Yaskawa INFORM job: BATMAN_ALL.JBI

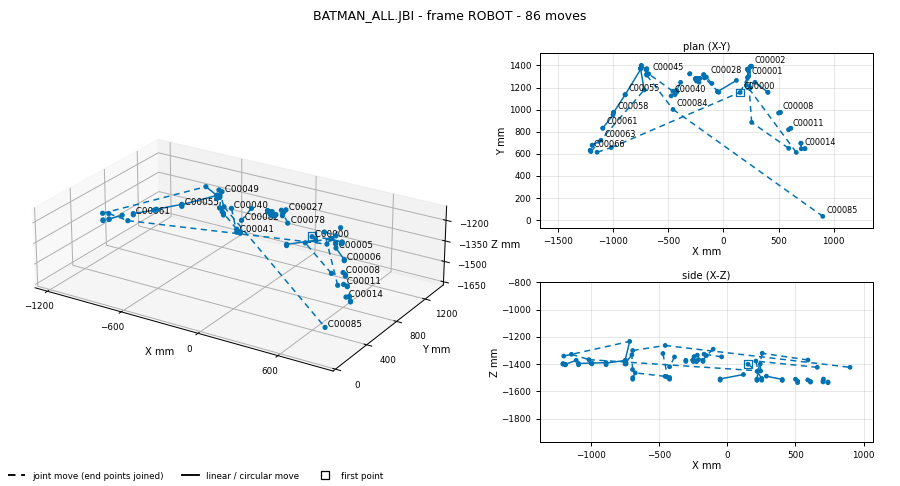
[picture p0: tool path of BATMAN_ALL.JBI in frame ROBOT, 86 of 157 moves have a stored position in this frame; points joined in program order, loops and branches not executed]
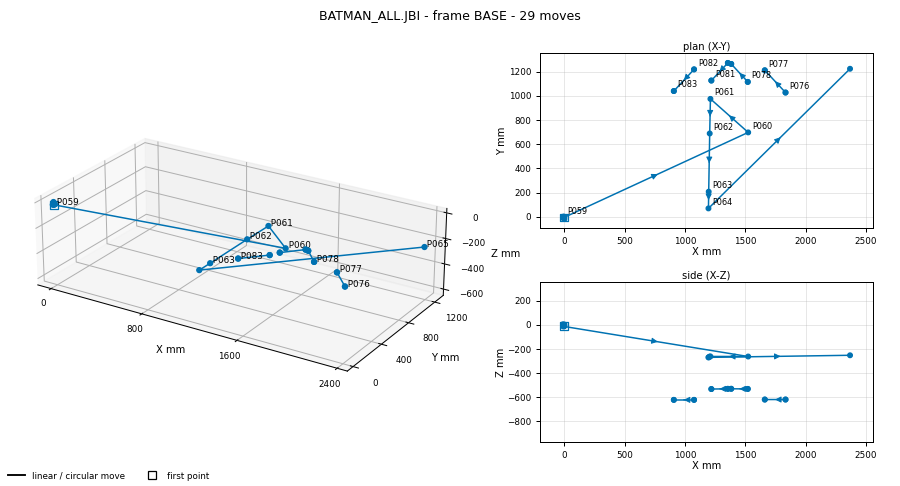
[picture p1: tool path of BATMAN_ALL.JBI in frame BASE, 29 of 157 moves have a stored position in this frame; points joined in program order, loops and branches not executed]
/JOB
//NAME BATMAN_ALL
///FOLDERNAME KRIS-SCIANA
//POS
///NPOS 86,86,0,38,0,0
///TOOL 0
///POSTYPE ROBOT
///RECTAN
///RCONF 0,0,0,0,0,0,0,0,0,0,0,0,0,0,0,0,0,0,0,0,0,0,0,0
C00000=152.410,1154.783,-1401.344,10.8585,26.8248,-46.4937
C00001=219.135,1290.433,-1453.397,13.1324,27.7106,-79.4132
C00002=252.850,1392.626,-1506.056,13.1307,27.7072,-79.4089
C00003=252.842,1392.620,-1508.783,13.1301,27.7068,-79.4080
C00004=252.850,1392.613,-1518.378,13.1306,27.7064,-79.4089
C00005=287.081,1247.667,-1488.936,13.1308,27.7079,-79.4066
C00006=403.589,1157.140,-1512.613,13.1304,27.7106,-79.4046
C00007=403.589,1157.122,-1519.985,13.1305,27.7097,-79.4043
C00008=500.680,969.258,-1511.018,13.1325,27.7074,-79.4005
C00009=516.044,974.881,-1524.930,13.1331,27.7092,-79.4004
C00010=516.045,974.868,-1535.811,13.1328,27.7077,-79.4001
C00011=590.606,818.366,-1515.976,13.1319,27.7058,-79.3988
C00012=610.782,831.337,-1527.481,13.1332,27.7070,-79.3997
C00013=610.774,831.333,-1532.290,13.1329,27.7070,-79.3992
C00014=705.770,645.699,-1509.934,13.1296,27.7061,-79.4018
C00015=702.820,695.837,-1524.665,13.1293,27.7044,-79.3984
C00016=702.809,695.833,-1530.916,13.1291,27.7040,-79.3963
C00017=738.969,646.930,-1531.718,13.1275,27.7068,-79.4007
C00018=738.965,646.937,-1536.801,13.1273,27.7075,-79.4010
C00019=592.006,649.855,-1370.263,13.1298,27.7033,-79.3961
C00020=256.954,884.347,-1320.582,10.9643,26.7399,-79.4986
C00021=226.416,1297.769,-1450.356,10.9643,26.7388,-15.7591
C00022=218.104,1365.766,-1510.694,4.6590,27.3838,-18.5852
C00023=218.092,1365.754,-1519.334,4.6575,27.3846,-18.5871
C00024=118.975,1264.663,-1476.628,4.6556,27.3863,-18.5969
C00025=-51.918,1162.894,-1508.930,4.6554,27.3843,-18.5935
C00026=-51.924,1162.893,-1518.207,4.6552,27.3847,-18.5926
C00027=-103.106,1236.815,-1291.023,4.6548,27.3832,-18.5938
C00028=-153.186,1294.382,-1337.444,-2.5810,29.3407,-40.5711
C00029=-177.451,1316.167,-1372.170,-2.5797,29.3412,-40.5749
C00030=-177.463,1316.142,-1380.653,-2.5821,29.3407,-40.5765
C00031=-210.259,1283.024,-1367.501,-2.5843,29.3397,-40.5838
C00032=-225.620,1283.017,-1376.307,-2.5829,29.3396,-40.5802
C00033=-225.613,1283.030,-1382.225,-2.5820,29.3397,-40.5809
C00034=-243.196,1259.338,-1345.105,-2.5829,29.3386,-40.5814
C00035=-253.627,1276.795,-1370.708,-2.5815,29.3400,-94.0341
C00036=-248.341,1281.400,-1375.363,-2.5806,29.3383,-94.0334
C00037=-248.343,1281.405,-1380.636,-2.5812,29.3384,-94.0354
C00038=-303.361,1324.266,-1372.348,-2.5804,29.3359,-94.0344
C00039=-303.363,1324.269,-1380.668,-2.5806,29.3358,-94.0352
C00040=-471.541,1124.138,-1322.421,-2.5821,29.3374,-94.0378
C00041=-436.993,1135.677,-1497.127,-2.5833,29.3385,-94.0377
C00042=-422.594,1159.988,-1498.740,-2.5814,29.3381,-94.0327
C00043=-422.595,1159.986,-1510.903,-2.5817,29.3385,-94.0330
C00044=-455.700,1166.055,-1490.114,-2.5799,29.3369,-94.0339
C00045=-674.596,1323.179,-1464.338,-2.5825,29.3370,-94.0343
C00046=-692.829,1369.142,-1499.740,-2.5956,29.3274,-94.0386
C00047=-692.829,1369.134,-1511.111,-2.5953,29.3273,-94.0360
C00048=-694.274,1320.333,-1440.373,-2.5948,29.3272,-94.0370
C00049=-699.144,1360.561,-1331.781,19.2113,25.3199,54.7614
C00050=-742.001,1399.272,-1388.079,19.2141,25.3197,54.7634
C00051=-742.001,1399.307,-1398.942,19.2156,25.3171,54.7657
C00052=-749.229,1371.947,-1375.142,19.2122,25.3194,54.7649
C00053=-749.245,1371.950,-1399.047,19.2137,25.3200,54.7650
C00054=-744.062,1371.872,-1373.000,19.2081,25.3216,54.7703
C00055=-888.177,1135.095,-1392.458,19.2114,25.3213,54.7713
C00056=-888.162,1135.097,-1404.947,19.2099,25.3206,54.7706
C00057=-888.146,1135.084,-1389.652,19.2087,25.3204,54.7704
C00058=-992.935,974.707,-1392.448,19.2118,25.3202,54.7709
C00059=-992.926,974.691,-1398.054,19.2108,25.3207,54.7707
C00060=-998.229,951.939,-1392.438,19.2128,25.3209,54.7710
C00061=-1090.439,832.216,-1395.757,19.2120,25.3253,54.7669
C00062=-1090.449,832.216,-1404.874,19.2124,25.3260,54.7666
C00063=-1107.538,722.615,-1372.300,19.2115,25.3258,54.7652
C00064=-1186.713,677.650,-1401.899,19.2118,25.3233,54.7691
C00065=-1186.711,677.656,-1405.576,19.2118,25.3228,54.7692
C00066=-1204.504,631.027,-1396.106,19.2134,25.3226,54.7707
C00067=-1204.501,631.029,-1401.004,19.2135,25.3224,54.7708
C00068=-1198.537,620.359,-1341.276,19.2108,25.3216,54.7720
C00069=-715.412,1179.070,-1233.819,19.2159,25.3335,54.7762
C00070=-749.229,1371.947,-1375.142,19.2122,25.3194,54.7649
C00071=-1142.143,614.362,-1328.458,18.1291,25.2802,54.3071
C00072=-1014.182,656.385,-1367.467,19.2126,25.3035,24.7793
C00073=244.678,1197.356,-1450.442,14.1934,24.5334,-60.4282
C00074=242.567,1385.701,-1399.440,12.9652,27.2001,-79.4839
C00075=660.569,613.161,-1423.808,13.1448,27.7005,-139.3923
C00076=210.374,1220.455,-1377.909,14.2177,19.9635,-61.8713
C00077=226.382,1351.810,-1450.861,14.2179,19.9642,-61.8758
C00078=-41.244,1157.338,-1346.763,4.6551,27.3861,-18.5879
C00079=-169.787,1287.439,-1327.342,-2.5927,29.3373,-40.6168
C00080=-219.530,1247.683,-1334.789,-2.5902,29.3364,-82.5753
C00081=-386.471,1247.154,-1347.732,14.2186,19.9661,-61.8751
C00082=-422.753,1176.097,-1419.836,-2.5966,29.3308,-94.0443
C00083=-692.993,1311.701,-1300.606,-2.6070,29.3169,-94.0355
C00084=-454.695,1001.750,-1263.493,10.2829,30.0776,-90.6322
C00085=900.646,33.952,-1423.808,13.1448,27.7005,179.8982
BC00000=1473.101,32.856,1458.546
BC00001=1602.629,32.856,1262.258
BC00002=1602.629,32.863,1262.252
BC00003=1602.629,32.863,1262.252
BC00004=1602.629,32.863,1262.252
BC00005=1602.629,32.863,1262.252
BC00006=1602.629,32.863,1262.248
BC00007=1602.629,32.863,1262.248
BC00008=1602.629,32.863,1262.248
BC00009=1602.629,32.863,1262.248
BC00010=1602.629,32.863,1262.248
BC00011=1602.629,32.863,1262.248
BC00012=1602.629,32.863,1262.248
BC00013=1602.629,32.863,1262.248
BC00014=1602.629,32.863,1262.248
BC00015=1602.629,32.863,1262.248
BC00016=1602.629,32.863,1262.248
BC00017=1602.629,32.863,1262.248
BC00018=1602.629,32.863,1262.248
BC00019=1602.629,32.863,1262.248
BC00020=1602.629,32.863,1262.248
BC00021=1602.629,32.863,1262.248
BC00022=1602.629,32.863,1262.248
BC00023=1602.629,32.863,1262.248
BC00024=1602.629,32.863,1262.248
BC00025=1602.629,32.863,1262.248
BC00026=1602.629,32.863,1262.248
BC00027=1602.629,32.863,1262.248
BC00028=1602.629,32.863,1262.248
BC00029=1602.629,32.863,1262.248
BC00030=1602.629,32.863,1262.248
BC00031=1602.629,32.863,1262.248
BC00032=1602.629,32.863,1262.248
BC00033=1602.629,32.863,1262.248
BC00034=1602.629,32.863,1262.248
BC00035=1602.629,32.863,1262.248
BC00036=1602.629,32.863,1262.248
BC00037=1602.629,32.863,1262.248
BC00038=1602.629,32.863,1262.248
BC00039=1602.629,32.863,1262.248
BC00040=1602.629,32.863,1262.248
BC00041=1602.629,32.863,1262.248
BC00042=1602.629,32.863,1262.248
BC00043=1602.629,32.863,1262.248
BC00044=1602.629,32.863,1262.248
BC00045=1602.629,32.863,1262.248
BC00046=1602.623,32.869,1262.243
BC00047=1602.623,32.869,1262.243
BC00048=1602.623,32.869,1262.243
BC00049=1602.629,32.850,1148.408
BC00050=1602.629,32.850,1148.408
BC00051=1602.629,32.850,1148.408
BC00052=1602.629,32.850,1148.408
BC00053=1602.629,32.850,1148.408
BC00054=1602.629,32.850,1148.408
BC00055=1602.629,32.850,1148.408
BC00056=1602.629,32.850,1148.408
BC00057=1602.629,32.850,1148.408
BC00058=1602.629,32.850,1148.408
BC00059=1602.629,32.850,1148.408
BC00060=1602.629,32.850,1148.408
BC00061=1602.629,32.850,1148.408
BC00062=1602.629,32.850,1148.408
BC00063=1602.629,32.850,1148.408
BC00064=1602.629,32.850,1148.408
BC00065=1602.629,32.850,1148.408
BC00066=1602.629,32.850,1148.408
BC00067=1602.629,32.850,1148.408
BC00068=1602.629,32.850,1148.408
BC00069=1602.629,32.856,1148.402
BC00070=1602.629,32.850,1148.408
BC00071=1602.629,32.850,1148.408
BC00072=1602.629,32.856,1527.186
BC00073=1602.629,32.856,1413.595
BC00074=1602.629,32.863,1262.252
BC00075=1602.629,32.863,1262.252
BC00076=1602.629,32.863,1262.252
BC00077=1602.629,32.863,1262.252
BC00078=1602.629,32.863,1262.252
BC00079=1602.629,32.863,1262.252
BC00080=1602.629,32.863,1262.252
BC00081=1602.629,32.863,1262.252
BC00082=1602.629,32.863,1262.252
BC00083=1602.629,32.863,1262.252
BC00084=1602.629,32.863,1262.252
BC00085=899.093,32.863,1856.752
///POSTYPE BASE
P00059=-2.448,-6.714,-12.718,0.0000,0.0000,0.0000
P00060=1524.284,698.404,-261.973,-0.4635,36.8346,-1.2388
P00061=1211.499,975.999,-261.374,0.5148,35.2356,175.5099
P00062=1205.574,689.500,-262.704,0.5159,35.2461,175.5270
P00063=1197.217,207.358,-268.729,0.4863,35.2395,175.4586
P00064=1195.199,68.975,-269.171,0.5092,35.2366,175.4908
P00065=2367.684,1225.356,-251.745,0.6375,35.5356,-175.5535
P00070=2.449,-18.318,2.615,0.0000,0.0000,0.0000
P00071=-2.048,-0.034,-9.092,0.0000,0.0000,0.0000
P00072=-1.595,-0.049,-6.373,0.0000,0.0000,0.0000
P00073=-8.474,-10.331,-11.894,0.0000,0.0000,0.0000
P00074=1.731,-3.007,-10.460,0.0000,0.0000,0.0000
///RCONF 0,1,0,0,0,0,0,0,0,0,0,0,0,0,0,0,0,0,0,0,0,0,0,0
P00075=-9.634,0.014,4.922,0.0000,0.0000,0.0000
///RCONF 0,0,0,0,0,0,0,0,0,0,0,0,0,0,0,0,0,0,0,0,0,0,0,0
P00076=1833.500,1028.615,-618.215,10.0256,37.5190,56.2681
P00077=1661.766,1212.555,-618.325,10.0309,37.5577,56.2858
P00078=1520.740,1116.757,-530.271,10.0398,37.5578,56.2925
P00079=1383.754,1265.334,-529.217,10.0293,37.5461,56.2787
P00080=1355.833,1273.708,-529.583,10.0283,37.5305,126.4716
P00081=1219.184,1127.874,-531.327,10.0137,37.5345,126.4324
P00082=1075.995,1220.294,-620.895,10.0203,37.5289,126.4576
P00083=908.434,1040.970,-620.895,10.0141,37.5419,126.4584
P00098=-1.000,0.000,-2.000,0.0000,0.0000,-60.0000
P00099=-10.497,4.418,3.734,0.0000,0.0000,0.0000
P00105=-13.000,6.000,-2.500,0.0000,0.0000,0.0000
P00106=13.000,-13.000,-3.000,0.0000,0.0000,0.0000
P00107=-12.000,8.000,-3.000,0.0000,0.0000,0.0000
P00108=0.000,0.000,-3.000,0.0000,0.0000,0.0000
P00110=13.000,10.000,-3.000,0.0000,0.0000,0.0000
P00111=-15.000,-15.000,-2.000,0.0000,0.0000,0.0000
P00112=15.000,7.000,-2.500,0.0000,0.0000,0.0000
P00113=-8.000,-10.000,-3.000,0.0000,0.0000,0.0000
P00114=10.000,-8.000,-3.000,0.0000,0.0000,0.0000
P00124=0.000,50.000,0.000,0.0000,0.0000,0.0000
P00125=0.000,0.000,2.400,0.0000,0.0000,0.0000
P00126=-50.000,0.000,0.000,0.0000,0.0000,0.0000
P00127=50.000,0.000,0.000,0.0000,0.0000,0.0000
P00170=4.000,4.000,-1.000,-10.0000,10.0000,-30.0000
P00171=-8.000,11.000,-2.000,0.0000,0.0000,-60.0000
//INST
///DATE 2024/02/20 09:55
///COMM NOWY SEARCH
///ATTR SC,RW,RJ
////FRAME ROBOT
///GROUP1 RB1,BS1
NOP
SFTOF
CALL JOB:ONLYCUT-R1_LONG
MOVJ C00000 BC00000 VJ=15.00
MOVJ C00001 BC00001 VJ=15.00
'POMIAR PRAWA STRONA
MOVL C00002 BC00002 V=250.0
'1
MOVL C00003 BC00003 V=166.7
MOVL C00004 BC00004 V=16.7 PL=0 SRCH RIN#(1)=ON T=1.00 DIS=20.0
TIMER T=0.20
IMOV P125 V=13.3 PL=0
TIMER T=0.20
IMOV P127 V=13.3 PL=0 SRCH RIN#(1)=ON DIS=20.0
TIMER T=0.20
GETS PX070 $PX001
TIMER T=0.10
MOVJ C00005 BC00005 VJ=15.00
'2
MOVL C00006 BC00006 V=50.0
MOVL C00007 BC00007 V=16.7 PL=0 SRCH RIN#(1)=ON T=1.00 DIS=20.0
TIMER T=0.20
IMOV P125 V=13.3 PL=0
TIMER T=0.20
IMOV P127 V=13.3 PL=0 SRCH RIN#(1)=ON DIS=20.0
TIMER T=0.20
GETS PX071 $PX001
TIMER T=0.10
MOVJ C00008 BC00008 VJ=15.00
'3
MOVL C00009 BC00009 V=50.0
MOVL C00010 BC00010 V=16.7 PL=0 SRCH RIN#(1)=ON T=1.00 DIS=20.0
TIMER T=0.20
IMOV P125 V=13.3 PL=0
TIMER T=0.20
IMOV P127 V=13.3 PL=0 SRCH RIN#(1)=ON DIS=20.0
TIMER T=0.20
GETS PX072 $PX001
TIMER T=0.10
MOVJ C00011 BC00011 VJ=15.00
'4
MOVL C00012 BC00012 V=50.0
MOVL C00013 BC00013 V=16.7 PL=0 SRCH RIN#(1)=ON T=1.00 DIS=20.0
TIMER T=0.20
IMOV P125 V=13.3 PL=0
TIMER T=0.20
IMOV P127 V=13.3 PL=0 SRCH RIN#(1)=ON DIS=20.0
TIMER T=0.20
GETS PX073 $PX001
TIMER T=0.10
MOVJ C00014 BC00014 VJ=15.00
'5
MOVL C00015 BC00015 V=50.0
MOVL C00016 BC00016 V=16.7 PL=0 SRCH RIN#(1)=ON T=1.00 DIS=20.0
TIMER T=0.20
IMOV P125 V=13.3 PL=0
TIMER T=0.20
IMOV P127 V=13.3 PL=0 SRCH RIN#(1)=ON DIS=20.0
TIMER T=0.20
GETS PX074 $PX001
TIMER T=0.10
MOVL C00017 BC00017 V=50.0
MOVL C00018 BC00018 V=16.7 PL=0 SRCH RIN#(1)=ON T=1.00 DIS=20.0
TIMER T=0.20
IMOV P125 V=13.3 PL=0
TIMER T=0.20
IMOV P127 V=13.3 PL=0 SRCH RIN#(1)=ON DIS=20.0
TIMER T=0.20
GETS PX075 $PX001
TIMER T=0.10
MOVJ C00019 BC00019 VJ=15.00
MOVJ C00020 BC00020 VJ=30.00
'POMIAR BATMAN
MOVJ C00021 BC00021 VJ=30.00
MOVL C00022 BC00022 V=166.7
MOVL C00023 BC00023 V=13.3 PL=0 SRCH RIN#(1)=ON T=1.00 DIS=20.0
TIMER T=0.20
IMOV P125 V=13.3 PL=0
TIMER T=0.20
IMOV P124 V=13.3 PL=0 SRCH RIN#(1)=ON DIS=20.0
TIMER T=0.20
GETS PX076 $PX001
TIMER T=0.10
MOVJ C00024 BC00024 VJ=30.00
MOVL C00025 BC00025 V=166.7
MOVL C00026 BC00026 V=16.7 PL=0 SRCH RIN#(1)=ON T=1.00 DIS=20.0
TIMER T=0.20
IMOV P125 V=13.3 PL=0
TIMER T=0.20
IMOV P124 V=13.3 PL=0 SRCH RIN#(1)=ON DIS=20.0
TIMER T=0.20
GETS PX077 $PX001
TIMER T=0.10
MOVJ C00027 BC00027 VJ=30.00
MOVJ C00028 BC00028 VJ=30.00
MOVL C00029 BC00029 V=166.7
MOVL C00030 BC00030 V=16.7 PL=0 SRCH RIN#(1)=ON T=1.00 DIS=20.0
TIMER T=0.20
IMOV P125 V=13.3 PL=0
TIMER T=0.20
IMOV P124 V=13.3 PL=0 SRCH RIN#(1)=ON DIS=20.0
TIMER T=0.20
GETS PX078 $PX001
TIMER T=0.10
MOVJ C00031 BC00031 VJ=30.00
MOVL C00032 BC00032 V=166.7
MOVL C00033 BC00033 V=16.7 PL=0 SRCH RIN#(1)=ON T=1.00 DIS=20.0
TIMER T=0.20
IMOV P125 V=13.3 PL=0
TIMER T=0.20
IMOV P124 V=13.3 PL=0 SRCH RIN#(1)=ON DIS=20.0
TIMER T=0.20
GETS PX079 $PX001
TIMER T=0.10
MOVJ C00034 BC00034 VJ=30.00
MOVJ C00035 BC00035 VJ=30.00
MOVL C00036 BC00036 V=166.7
MOVL C00037 BC00037 V=16.7 PL=0 SRCH RIN#(1)=ON T=1.00 DIS=20.0
TIMER T=0.20
IMOV P125 V=13.3 PL=0
TIMER T=0.20
IMOV P124 V=13.3 PL=0 SRCH RIN#(1)=ON DIS=20.0
TIMER T=0.20
GETS PX080 $PX001
TIMER T=0.10
MOVL C00038 BC00038 V=166.7
MOVL C00039 BC00039 V=16.7 PL=0 SRCH RIN#(1)=ON T=1.00 DIS=20.0
TIMER T=0.20
IMOV P125 V=13.3 PL=0
TIMER T=0.20
IMOV P124 V=13.3 PL=0 SRCH RIN#(1)=ON DIS=20.0
TIMER T=0.20
GETS PX081 $PX001
TIMER T=0.10
MOVJ C00040 BC00040 VJ=30.00
MOVJ C00041 BC00041 VJ=30.00
MOVL C00042 BC00042 V=166.7
MOVL C00043 BC00043 V=16.7 PL=0 SRCH RIN#(1)=ON T=1.00 DIS=20.0
TIMER T=0.20
IMOV P125 V=13.3 PL=0
TIMER T=0.20
IMOV P124 V=13.3 PL=0 SRCH RIN#(1)=ON DIS=20.0
TIMER T=0.20
GETS PX082 $PX001
TIMER T=0.10
MOVJ C00044 BC00044 VJ=15.00
MOVJ C00045 BC00045 VJ=30.00
MOVL C00046 BC00046 V=166.7
MOVL C00047 BC00047 V=16.7 PL=0 SRCH RIN#(1)=ON T=1.00 DIS=20.0
TIMER T=0.20
IMOV P125 V=23.0 PL=0
TIMER T=0.20
IMOV P124 V=23.0 PL=0 SRCH RIN#(1)=ON DIS=20.0
TIMER T=0.20
GETS PX083 $PX001
TIMER T=0.10
MOVJ C00048 BC00048 VJ=30.00
'KONIEC POMIAR BATMAN 1STR
SFTOF
MOVJ C00049 BC00049 VJ=15.00
'1
MOVL C00050 BC00050 V=166.7
MOVL C00051 BC00051 V=16.7 PL=0 SRCH RIN#(1)=ON T=1.00 DIS=20.0
TIMER T=0.20
IMOV P125 V=13.3 PL=0
TIMER T=0.20
IMOV P126 V=13.3 PL=0 SRCH RIN#(1)=ON DIS=20.0
TIMER T=0.20
GETS PX059 $PX001
TIMER T=0.10
MOVL C00052 BC00052 V=166.7
MOVL C00053 BC00053 V=16.7 PL=0 SRCH RIN#(1)=ON T=1.00 DIS=20.0
TIMER T=0.20
IMOV P125 V=13.3 PL=0
TIMER T=0.20
IMOV P126 V=13.3 PL=0 SRCH RIN#(1)=ON DIS=20.0
TIMER T=0.20
GETS PX060 $PX001
TIMER T=0.10
MOVJ C00054 BC00054 VJ=0.78
'2
MOVL C00055 BC00055 V=50.0
MOVL C00056 BC00056 V=16.7 PL=0 SRCH RIN#(1)=ON T=1.00 DIS=20.0
TIMER T=0.20
IMOV P125 V=13.3 PL=0
TIMER T=0.20
IMOV P126 V=13.3 PL=0 SRCH RIN#(1)=ON DIS=20.0
TIMER T=0.20
GETS PX061 $PX001
TIMER T=0.10
MOVJ C00057 BC00057 VJ=0.78
'3
MOVL C00058 BC00058 V=50.0
MOVL C00059 BC00059 V=16.7 PL=0 SRCH RIN#(1)=ON T=1.00 DIS=20.0
TIMER T=0.20
IMOV P125 V=13.3 PL=0
TIMER T=0.20
IMOV P126 V=13.3 PL=0 SRCH RIN#(1)=ON DIS=20.0
TIMER T=0.20
GETS PX062 $PX001
TIMER T=0.10
MOVJ C00060 BC00060 VJ=0.78
'4
MOVL C00061 BC00061 V=50.0
MOVL C00062 BC00062 V=16.7 PL=0 SRCH RIN#(1)=ON T=1.00 DIS=20.0
TIMER T=0.20
IMOV P125 V=13.3 PL=0
TIMER T=0.20
IMOV P126 V=13.3 PL=0 SRCH RIN#(1)=ON DIS=20.0
TIMER T=0.20
GETS PX063 $PX001
TIMER T=0.10
MOVJ C00063 BC00063 VJ=30.00
'5
MOVL C00064 BC00064 V=50.0
MOVL C00065 BC00065 V=16.7 PL=0 SRCH RIN#(1)=ON T=1.00 DIS=20.0
TIMER T=0.20
IMOV P125 V=13.3 PL=0
TIMER T=0.20
IMOV P126 V=13.3 PL=0 SRCH RIN#(1)=ON DIS=20.0
TIMER T=0.20
GETS PX064 $PX001
TIMER T=0.10
MOVL C00066 BC00066 V=50.0
MOVL C00067 BC00067 V=16.7 PL=0 SRCH RIN#(1)=ON T=1.00 DIS=20.0
TIMER T=0.20
IMOV P125 V=13.3 PL=0
TIMER T=0.20
IMOV P126 V=13.3 PL=0 SRCH RIN#(1)=ON DIS=20.0
TIMER T=0.20
GETS PX065 $PX001
TIMER T=0.10
MOVJ C00068 BC00068 VJ=15.00
'********
'********
'********
MOVJ C00069 BC00069 VJ=15.00
MOVL C00070 BC00070 V=333.3
MACRO1 MJ#(0) ARGF7
SFTOF
SFTON P170
MOVL P059 V=83.3
ARCON
SFTOF
SFTON P099
MOVL P060 V=10.8
MOVL P061 V=10.8
MOVL P062 V=10.8
MOVL P063 V=10.8
MOVL P064 V=10.8
MOVL P065 V=10.8
ARCOF
MOVJ C00071 BC00071 VJ=15.00
SFTOF
MOVJ C00072 BC00072 VJ=15.00
MOVJ C00073 BC00073 VJ=15.00
SFTON P171
MOVJ C00074 BC00074 VJ=15.00
MOVL P070 V=83.3
ARCON
SFTOF
SFTON P098
MOVL P071 V=10.8
MOVL P072 V=10.8
MOVL P073 V=10.8
MOVL P074 V=10.8
MOVL P075 V=10.8
ARCOF
SFTOF
MOVJ C00075 BC00075 VJ=15.00
MOVJ C00076 BC00076 VJ=30.00
MOVJ C00077 BC00077 VJ=30.00
SFTON P110
MOVL P076 V=83.3
SFTOF
ARCON
SFTON P108
MOVL P076 V=10.8
MOVL P077 V=10.8
SFTON P111
MOVL P077 V=10.8
ARCOF
SFTOF
MOVJ C00078 BC00078 VJ=30.00
MOVJ C00079 BC00079 VJ=30.00
SFTON P112
MOVL P078 V=83.3
ARCON
SFTOF
SFTON P108
MOVL P078 V=10.8
MOVL P079 V=10.8
SFTOF
SFTON P113
MOVL P079 V=10.8
ARCOF
SFTOF
MOVJ C00080 BC00080 VJ=30.00
SFTON P114
MOVL P080 V=83.3
SFTOF
ARCON
SFTON P108
MOVL P080 V=10.8
MOVL P081 V=10.8
SFTOF
SFTON P105
MOVL P081 V=10.8
SFTOF
ARCOF
MOVJ C00081 BC00081 VJ=30.00
MOVJ C00082 BC00082 VJ=30.00
SFTON P106
MOVL P082 V=83.3
SFTOF
ARCON
SFTON P108
MOVL P082 V=10.8
MOVL P083 V=10.8
SFTOF
SFTON P107
MOVL P083 V=10.8
SFTOF
ARCOF
MOVJ C00083 BC00083 VJ=30.00
MOVJ C00084 BC00084 VJ=30.00
MOVJ C00085 BC00085 VJ=30.00
CALL JOB:ONLYCUT-R1_LONG
END
